FUNCTION_BLOCK FB_ConfigControlJson EXTENDS FB_JsonSchemaEx_OLD
VAR_INPUT
END_VAR
VAR_OUTPUT
	P_sJsonid			: MPM_JsonParser.DUT_JsonSchema := (member := '_id', typeClass := E_TypeClassEx.TYPE_STRING,jsonValueRoot := jsonRoot);
	P_sJsonTimeStamp	: MPM_JsonParser.DUT_JsonSchema := (member := 'time_stamp', typeClass := E_TypeClassEx.TYPE_FILETIME,jsonValueRoot := jsonRoot);		
	P_sJsonRecipe		: MPM_JsonParser.DUT_JsonSchema := (member := 'Recipe', typeClass := E_TypeClassEx.TYPE_JSON,jsonValueRoot := jsonRoot);
	P_sJsonSystem		: MPM_JsonParser.DUT_JsonSchema := (member := 'System', typeClass := E_TypeClassEx.TYPE_JSON,jsonValueRoot := jsonRoot);
	P_sJsonIOValues		: MPM_JsonParser.DUT_JsonSchema := (member := 'IO', typeClass := E_TypeClassEx.TYPE_JSON,jsonValueRoot := jsonRoot);
END_VAR
VAR
	jsonRoot : SJsonValue;	
END_VAR

METHOD PUBLIC  M_CreateSchemaJson : BOOL
VAR_IN_OUT
END_VAR
VAR
	
END_VAR
jsonRoot := THIS^.NewDocument();
M_SetJsonSchema(jsonRoot,P_sJsonid);
M_SetJsonSchema(jsonRoot,P_sJsonRecipe);
M_SetJsonSchema(jsonRoot,P_sJsonSystem);
M_SetJsonSchema(jsonRoot,P_sJsonIOValues);
M_SetJsonSchema(jsonRoot,P_sJsonTimeStamp);
END_METHOD

METHOD PUBLIC  M_PraseSchemaJson : BOOL
VAR_INPUT
END_VAR
jsonRoot := THIS^.GetDocumentRoot();
IF jsonRoot > 0 THEN
	M_PraseJsonSchema(jsonRoot,P_sJsonid);
	M_PraseJsonSchema(jsonRoot,P_sJsonRecipe);
	M_PraseJsonSchema(jsonRoot,P_sJsonSystem);
	M_PraseJsonSchema(jsonRoot,P_sJsonIOValues);
	M_PraseJsonSchema(jsonRoot,P_sJsonTimeStamp);
END_IF
END_METHOD

END_FUNCTION_BLOCK

(* stored: Version 1.1.0.1, ProductVersion 3.1.4024.12
   POU FB_ConfigControlJson: Id {fd6fc35a-3532-4b43-8957-b75eb939e4ec}, SpecialFunc None
   Method M_CreateSchemaJson: Id {7317fc8b-58ff-4f51-8cc3-8f88c1719a9d}
   Method M_PraseSchemaJson: Id {664025a6-1001-4bee-b12f-66995b59e06c} *)
